(* PLC project hvs_2c_loc_cb_mgt, GEENSOFT ControlBuild 2010-3c *)
(* stored: creationDateTime 2011-09-19T16:15:47-01:00 *)

PROGRAM hvs.hvs_2c_loc_cb_mgt
  VAR_INPUT
    ILvViuDjIsPt : BOOL := false;
    ILvViuDjSiQlmCcTfp : BOOL := false;
    ILvViuDjc1 : BOOL := false;
    ILvViuDjc2 : BOOL := false;
    ILvViuDjm : BOOL := false;
    ILvViuNoSuriDjc1 : BOOL := false;
    ILvViuNoSuriDjc2 : BOOL := false;
    ILvViuQD : BOOL := false;
  END_VAR
  VAR_INPUT
    C1_Hvs_ICbCntrReload : INT := 0;
    C2_Hvs_ICbCntrReload : INT := 0;
    C3_Hvs_ICbCntrReload : INT := 0;
    C4_Hvs_ICbCntrReload : INT := 0;
  END_VAR
  VAR_INPUT
    Air_IAuxCompPressSwitch : BOOL := false;
    Atp_ICLHvOrdersSupprsd : BOOL := false;
    Atp_ICLOpengCb : BOOL := false;
    CL_Hvs_CCloseGenDj : BOOL := false;
    Omc_IConsistMode : BYTE := 0;
    Trc_IAuthCbc1 : BOOL := false;
    Trc_IAuthCbc2 : BOOL := false;
    Trc_IAuthCbm : BOOL := false;
  END_VAR
  VAR_INPUT
    PDelayBefReload : DINT := 1000;
    PDelayOpengCb : DINT := 1000;
    PDelayOpengOvercurrent : DINT := 300;
    PDurationPulseCloseCb : DINT := 500;
    PReloadTrainLimit : INT := 3;
    PTimeOutPcoDj : DINT := 30000;
    PTimeOutReload : INT := 300;
  END_VAR
  VAR_INPUT
    Hvs_FVc2CritFaultTfp : BOOL := false;
    Hvs_FVe1CritFaultTfp : BOOL := false;
    Hvs_FVe2CritFaultTfp : BOOL := false;
    Hvs_FVi2CritFaultTfp : BOOL := false;
    Hvs_FViuCritFaultTfp1 : BOOL := false;
    Hvs_FViuCritFaultTfp2 : BOOL := false;
    Hvs_IHocDC : BOOL := false;
    Hvs_IHocGround : BOOL := false;
    Hvs_IModeElec : BOOL := false;
    Hvs_IPntDown : BOOL := false;
    Hvs_IPntDownAc : BOOL := false;
    Hvs_IPntDownDc : BOOL := false;
    Hvs_IPresCatSelected : BOOL := false;
    Hvs_IPresMonoCat : BOOL := false;
    IHoldDjQtSoft : BOOL := false;
    IOvercurrentQlm : BOOL := false;
    IPcoElec : BOOL := false;
    IPcoPntFinished : BOOL := false;
    IPntRaisedAc : BOOL := false;
    IPntRaisedDc : BOOL := false;
    ITrBrManipAuth : BOOL := false;
  END_VAR
  VAR_OUTPUT
    CLvViuCloseDj1 : BOOL := false;
    CLvViuCloseDj2 : BOOL := false;
    CLvViuDjC1 : BOOL := false;
    CLvViuDjC2 : BOOL := false;
    CLvViuDjM : BOOL := false;
  END_VAR
  VAR_OUTPUT
    Hvs_FViuDjC1 : BOOL := false;
    Hvs_FViuDjC2 : BOOL := false;
    Hvs_FViuDjM : BOOL := false;
    Hvs_ICbCntrReload : INT := 0;
    Hvs_ISyncStateDjC1 : BYTE := 0;
    Hvs_ISyncStateDjC2 : BYTE := 0;
    Hvs_ISyncStateDjM : BYTE := 0;
    Hvs_IViuDjC1Isold : BOOL := false;
    Hvs_IViuDjC2Isold : BOOL := false;
    Hvs_IViuDjMIsold : BOOL := false;
    IAllCbClosed : BOOL := false;
    IOpengCbReqstdDjC1 : BOOL := false;
    IOpengCbReqstdDjC2 : BOOL := false;
    IOpengCbReqstdDjM : BOOL := false;
    IPcoCbFailure : BOOL := false;
    ISumAuthCloseCb : DINT := 0;
    ISumAvailCb : DINT := 0;
    ISumRemaingCb : DINT := 0;
  END_VAR

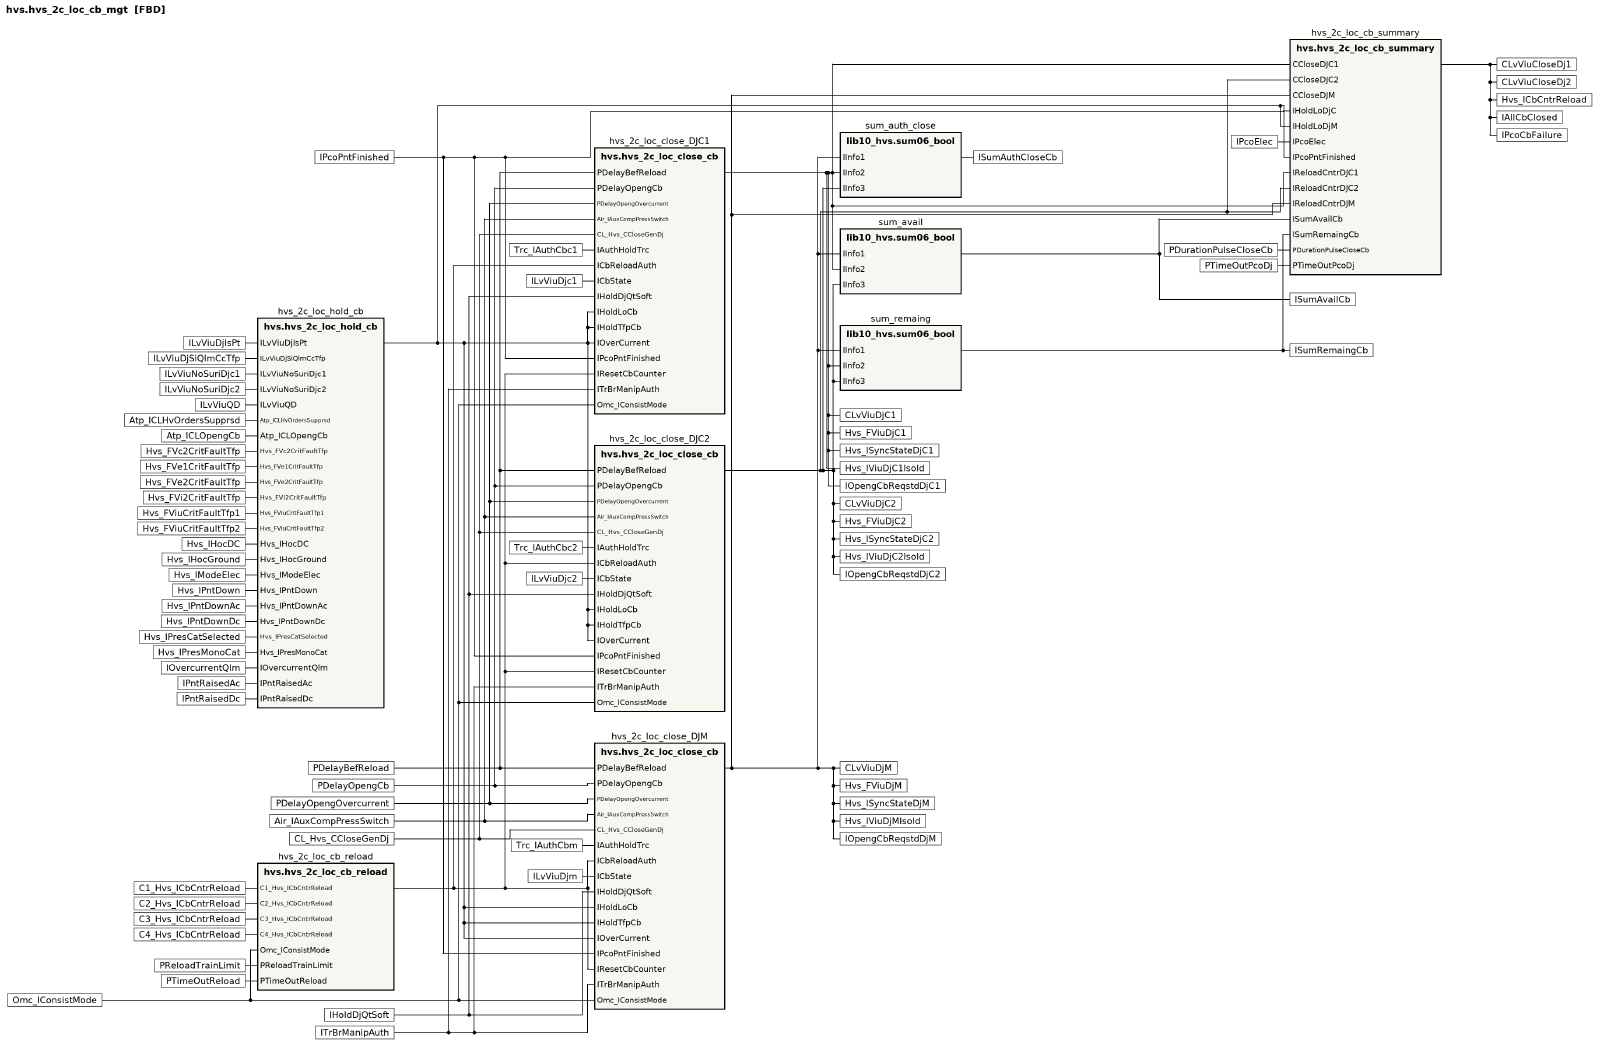
(* FBD diagram, written out as Structured Text *)
hvs_2c_loc_cb_reload(C1_Hvs_ICbCntrReload := C1_Hvs_ICbCntrReload, C2_Hvs_ICbCntrReload := C2_Hvs_ICbCntrReload, C3_Hvs_ICbCntrReload := C3_Hvs_ICbCntrReload, C4_Hvs_ICbCntrReload := C4_Hvs_ICbCntrReload, Omc_IConsistMode := Omc_IConsistMode, PReloadTrainLimit := PReloadTrainLimit, PTimeOutReload := PTimeOutReload);
hvs_2c_loc_hold_cb(ILvViuDjIsPt := ILvViuDjIsPt, ILvViuDjSiQlmCcTfp := ILvViuDjSiQlmCcTfp, ILvViuNoSuriDjc1 := ILvViuNoSuriDjc1, ILvViuNoSuriDjc2 := ILvViuNoSuriDjc2, ILvViuQD := ILvViuQD, Atp_ICLHvOrdersSupprsd := Atp_ICLHvOrdersSupprsd, Atp_ICLOpengCb := Atp_ICLOpengCb, Hvs_FVc2CritFaultTfp := Hvs_FVc2CritFaultTfp, Hvs_FVe1CritFaultTfp := Hvs_FVe1CritFaultTfp, Hvs_FVe2CritFaultTfp := Hvs_FVe2CritFaultTfp, Hvs_FVi2CritFaultTfp := Hvs_FVi2CritFaultTfp, Hvs_FViuCritFaultTfp1 := Hvs_FViuCritFaultTfp1, Hvs_FViuCritFaultTfp2 := Hvs_FViuCritFaultTfp2, Hvs_IHocDC := Hvs_IHocDC, Hvs_IHocGround := Hvs_IHocGround, Hvs_IModeElec := Hvs_IModeElec, Hvs_IPntDown := Hvs_IPntDown, Hvs_IPntDownAc := Hvs_IPntDownAc, Hvs_IPntDownDc := Hvs_IPntDownDc, Hvs_IPresCatSelected := Hvs_IPresCatSelected, Hvs_IPresMonoCat := Hvs_IPresMonoCat, IOvercurrentQlm := IOvercurrentQlm, IPntRaisedAc := IPntRaisedAc, IPntRaisedDc := IPntRaisedDc);
hvs_2c_loc_close_DJM(PDelayBefReload := PDelayBefReload, PDelayOpengCb := PDelayOpengCb, PDelayOpengOvercurrent := PDelayOpengOvercurrent, Air_IAuxCompPressSwitch := Air_IAuxCompPressSwitch, CL_Hvs_CCloseGenDj := CL_Hvs_CCloseGenDj, IAuthHoldTrc := Trc_IAuthCbm, ICbReloadAuth := hvs_2c_loc_cb_reload.ICbReloadAuth, ICbState := ILvViuDjm, IHoldDjQtSoft := IHoldDjQtSoft, IHoldLoCb := hvs_2c_loc_hold_cb.IHoldLoDjM, IHoldTfpCb := hvs_2c_loc_hold_cb.IHoldTfpDjM, IOverCurrent := hvs_2c_loc_hold_cb.IOverCurrentDjM, IPcoPntFinished := IPcoPntFinished, IResetCbCounter := hvs_2c_loc_cb_reload.IResetCbCounter, ITrBrManipAuth := ITrBrManipAuth, Omc_IConsistMode := Omc_IConsistMode);
CLvViuDjM := hvs_2c_loc_close_DJM.CCbKeptOpend;
hvs_2c_loc_close_DJC1(PDelayBefReload := PDelayBefReload, PDelayOpengCb := PDelayOpengCb, PDelayOpengOvercurrent := PDelayOpengOvercurrent, Air_IAuxCompPressSwitch := Air_IAuxCompPressSwitch, CL_Hvs_CCloseGenDj := CL_Hvs_CCloseGenDj, IAuthHoldTrc := Trc_IAuthCbc1, ICbReloadAuth := hvs_2c_loc_cb_reload.ICbReloadAuth, ICbState := ILvViuDjc1, IHoldDjQtSoft := IHoldDjQtSoft, IHoldLoCb := hvs_2c_loc_hold_cb.IHoldLoDjC, IHoldTfpCb := hvs_2c_loc_hold_cb.IHoldTfpDjC1, IOverCurrent := hvs_2c_loc_hold_cb.IOverCurrentDjC1, IPcoPntFinished := IPcoPntFinished, IResetCbCounter := hvs_2c_loc_cb_reload.IResetCbCounter, ITrBrManipAuth := ITrBrManipAuth, Omc_IConsistMode := Omc_IConsistMode);
Hvs_FViuDjC1 := hvs_2c_loc_close_DJC1.FCbFault;
Hvs_IViuDjMIsold := hvs_2c_loc_close_DJM.ICbIsold;
CLvViuDjC1 := hvs_2c_loc_close_DJC1.CCbKeptOpend;
Hvs_FViuDjM := hvs_2c_loc_close_DJM.FCbFault;
Hvs_IViuDjC1Isold := hvs_2c_loc_close_DJC1.ICbIsold;
IOpengCbReqstdDjC1 := hvs_2c_loc_close_DJC1.IOpengCbReqstd;
hvs_2c_loc_close_DJC2(PDelayBefReload := PDelayBefReload, PDelayOpengCb := PDelayOpengCb, PDelayOpengOvercurrent := PDelayOpengOvercurrent, Air_IAuxCompPressSwitch := Air_IAuxCompPressSwitch, CL_Hvs_CCloseGenDj := CL_Hvs_CCloseGenDj, IAuthHoldTrc := Trc_IAuthCbc2, ICbReloadAuth := hvs_2c_loc_cb_reload.ICbReloadAuth, ICbState := ILvViuDjc2, IHoldDjQtSoft := IHoldDjQtSoft, IHoldLoCb := hvs_2c_loc_hold_cb.IHoldLoDjC, IHoldTfpCb := hvs_2c_loc_hold_cb.IHoldTfpDjC2, IOverCurrent := hvs_2c_loc_hold_cb.IOverCurrentDjC2, IPcoPntFinished := IPcoPntFinished, IResetCbCounter := hvs_2c_loc_cb_reload.IResetCbCounter, ITrBrManipAuth := ITrBrManipAuth, Omc_IConsistMode := Omc_IConsistMode);
sum_auth_close(IInfo1 := hvs_2c_loc_close_DJM.ICbAuthClose, IInfo2 := hvs_2c_loc_close_DJC1.ICbAuthClose, IInfo3 := hvs_2c_loc_close_DJC2.ICbAuthClose);
ISumAuthCloseCb := sum_auth_close.ISum;
Hvs_ISyncStateDjC1 := hvs_2c_loc_close_DJC1.ISyncStateDj;
sum_avail(IInfo1 := hvs_2c_loc_close_DJM.ICbAvail, IInfo2 := hvs_2c_loc_close_DJC1.ICbAvail, IInfo3 := hvs_2c_loc_close_DJC2.ICbAvail);
ISumAvailCb := sum_avail.ISum;
CLvViuDjC2 := hvs_2c_loc_close_DJC2.CCbKeptOpend;
Hvs_FViuDjC2 := hvs_2c_loc_close_DJC2.FCbFault;
Hvs_IViuDjC2Isold := hvs_2c_loc_close_DJC2.ICbIsold;
sum_remaing(IInfo1 := hvs_2c_loc_close_DJM.ICbRemaing, IInfo2 := hvs_2c_loc_close_DJC1.ICbRemaing, IInfo3 := hvs_2c_loc_close_DJC2.ICbRemaing);
ISumRemaingCb := sum_remaing.ISum;
IOpengCbReqstdDjC2 := hvs_2c_loc_close_DJC2.IOpengCbReqstd;
Hvs_ISyncStateDjC2 := hvs_2c_loc_close_DJC2.ISyncStateDj;
hvs_2c_loc_cb_summary(CCloseDJC1 := hvs_2c_loc_close_DJC1.CCbClose, CCloseDJC2 := hvs_2c_loc_close_DJC2.CCbClose, CCloseDJM := hvs_2c_loc_close_DJM.CCbClose, IHoldLoDjC := hvs_2c_loc_hold_cb.IHoldLoDjC, IHoldLoDjM := hvs_2c_loc_hold_cb.IHoldLoDjM, IPcoElec := IPcoElec, IPcoPntFinished := IPcoPntFinished, IReloadCntrDJC1 := hvs_2c_loc_close_DJC1.ICbReloadCntr, IReloadCntrDJC2 := hvs_2c_loc_close_DJC2.ICbReloadCntr, IReloadCntrDJM := hvs_2c_loc_close_DJM.ICbReloadCntr, ISumAvailCb := sum_avail.ISum, ISumRemaingCb := sum_remaing.ISum, PDurationPulseCloseCb := PDurationPulseCloseCb, PTimeOutPcoDj := PTimeOutPcoDj);
CLvViuCloseDj1 := hvs_2c_loc_cb_summary.CCloseCb1;
CLvViuCloseDj2 := hvs_2c_loc_cb_summary.CCloseCb2;
Hvs_ICbCntrReload := hvs_2c_loc_cb_summary.Hvs_ICbCntrReload;
IAllCbClosed := hvs_2c_loc_cb_summary.IAllCbClosed;
IPcoCbFailure := hvs_2c_loc_cb_summary.IPcoDjFailure;
IOpengCbReqstdDjM := hvs_2c_loc_close_DJM.IOpengCbReqstd;
Hvs_ISyncStateDjM := hvs_2c_loc_close_DJM.ISyncStateDj;
END_PROGRAM
